(*
SPDX-FileCopyrightText: © 2026 Oleksandr Tiutyk <trofimich@gmail.com>
SPDX-License-Identifier: MIT
License: https://opensource.org/license/mit
*)

{attribute 'no_explicit_call' := 'do not call this function block directly'} 
PROGRAM ExceptionHandlingPolicies
VAR
	{attribute 'hide'} 
	_ClassName : STRING := __POUNAME();
	
	{attribute 'hide'} 
	_SetErrorAndStop : SetErrorAndStopExceptionHandlingPolicy; 
	{attribute 'hide'} 
	_SetErrorAndContinue : SetErrorAndContinueExceptionHandlingPolicy; 
	{attribute 'hide'} 
	_Ignore : IgnoreExceptionHandlingPolicy; 
END_VAR

{attribute 'monitoring' := 'call'}
PROPERTY ClassName : REFERENCE TO STRING
GET
ClassName REF= _ClassName;
END_GET
END_PROPERTY

{attribute 'monitoring' := 'call'}
PROPERTY Ignore : IExceptionHandlingPolicy
GET
Ignore := _Ignore;
END_GET
END_PROPERTY

{attribute 'monitoring' := 'call'}
PROPERTY NamespaceName : REFERENCE TO STRING
GET
NamespaceName REF= CurrentNamespace.Name;
END_GET
END_PROPERTY

{attribute 'monitoring' := 'call'}
PROPERTY SetErrorAndContinue : IExceptionHandlingPolicy
GET
SetErrorAndContinue := _SetErrorAndContinue;
END_GET
END_PROPERTY

{attribute 'monitoring' := 'call'}
PROPERTY SetErrorAndStop : IExceptionHandlingPolicy
GET
SetErrorAndStop := _SetErrorAndStop;
END_GET
END_PROPERTY

END_PROGRAM

(* stored: Version 1.1.0.1
   POU ExceptionHandlingPolicies: Id {08b71951-ad97-44a8-b5cc-b262511b6f70}, SpecialFunc None
   Property ClassName: Id {304036be-83ce-436b-8796-8bb9a917572e}
   Get Get: Id {42386e35-a242-4e17-9672-f0bbcb69971b}
   Property Ignore: Id {3fa5ddfd-092f-465d-8780-b698a4f21208}
   Get Get: Id {c36611be-4c85-4425-9b88-214f05dfc532}
   Property NamespaceName: Id {04c6ab03-30ec-4b23-ba7c-1d680266d5e9}
   Get Get: Id {89fb96ad-ac34-4aec-bd0e-5deb929f57ef}
   Property SetErrorAndContinue: Id {fbd978c5-f856-4be6-9cd4-d181823679a3}
   Get Get: Id {a417abe0-3b26-4c31-afeb-59de23130f2f}
   Property SetErrorAndStop: Id {40adec1c-f262-4483-9cda-8640fb51ad5f}
   Get Get: Id {e4a92697-c94a-4d25-9e15-f39344eac26a} *)
